PROGRAM MAIN
VAR
 
 fbLineRegulator : SM_LineRegulator;
 fbSymbolPathStorage : SymbolPathStorage;

END_VAR

fbLineRegulator(
	 sSubscription1 := 'TL1Synch',
	 sSubscription2 := 'TL2Synch',
	 sSubscription3 := 'TL3Synch'
);

END_PROGRAM

(* stored: Version 1.1.0.1, ProductVersion 3.1.4024.2
   POU MAIN: Id {4a3c7469-a95d-43da-b36d-b6415d027575}, SpecialFunc None *)
